Staubli VAL3: Robot_pippeting.dtx

aio aiAngleInclinarPipieta = {link=E954DA08-7D0C-47C0-8458-4D7DB0686071}
aio aiNumAmpolla = {link=F94C03B3-E86B-41EA-9D21-23C2AFB25672}
aio aiNumBanyera = {link=3DE16CC9-CC25-4818-8F3E-A7F806CB7947}
aio aiNumPipeta = {link=5259214B-6548-4F3D-A189-73563EE6598D}
aio aiNumPlacaDosi = {link=C4FBE503-E51F-4D58-BE10-749D221ACEB2}
aio aiProgramaPlc = {link=8E5652B8-E4D3-4267-ADD0-9C5A815DF2D8}
aio aiWordComPlc = {link=5C2A04D3-4005-4B43-8647-C0FC7B49D3AE}
aio aiXOffset = {link=95067B68-557B-4170-88AF-FC9CF5B8ED7A}
aio aiYOffset = {link=396181D2-5171-4A97-9799-32514BBB5F95}
aio aiZApro = {link=2D158B67-9924-4741-B554-50FB73F41045}
aio aiZOffset = {link=7513B562-B4FE-4098-AA1C-29A8706B731C}
aio aoForceJ1 = {link=9B11B2FE-99BA-4B55-9ED8-E4037A61E514}
aio aoForceJ2 = {link=DFC528C5-C573-4C02-A89E-35D8A1151078}
aio aoForceJ3 = {link=EC117CCB-E5D8-4A5C-AB6E-61FBA1760A17}
aio aoForceJ4 = {link=24340562-5DCA-47E3-A269-832024611405}
aio aoForceJ5 = {link=DB01A7CB-9BAD-4D46-B614-A585779504D9}
aio aoForceJ6 = {link=7A496CE7-D747-4637-B99A-202C76C7E7CC}
aio aoProgramaRobot = {link=5113B9A1-604C-4D8B-9163-7217CBF800C7}
aio aoStatusRobot = {link=F45B1EFD-4428-4D7D-8172-ECCCA511584C}
aio aoTascaAlarma = {link=53CEF201-0BB5-4BE1-8271-49FFF55CF52D}
aio aoWordComRobot = {link=6DF138BB-5CBA-4ACE-9C62-0AC3DF2353CB}
aio aoWorkingMode = {link=F7E03293-48A3-4B69-9598-2FE8DDFE0186}
aio aoXActual = {link=7FC267A8-BFA4-4039-BDA4-9FB4B4F71D48}
aio aoYActual = {link=E23CA4B2-A08C-4C00-8E97-94551E73BB09}
aio aoZActual = {link=78A73075-60CA-4FDB-AFF0-231125481CE1}
aio aoZonaHome = {link=F5709703-FBB2-4816-9A2C-2FC6F0D8F434}
bool bNewLog
bool bPrimerCicle
bool bTaskDone
dio diAlarmaPlc = {link=E7921EDF-610C-4E3F-84A7-2F1F4421B713}
dio diMarxaMaquina = {link=C1F67030-A9C1-420C-9B9B-1F49F7080557}
dio diSafetyRearme = {link=5367EF22-1F58-447B-AD12-D8B84F185C6B}
dio doAlarmaColisioRobot = {link=EA8AD671-7535-4BE0-BEBB-B9246DF094E3}
dio doAlarmaTascaRobot = {link=FCAEE04F-32B9-421A-B1DD-A8CEAA94D1C9}
dio doRobotEnMoviment = {link=B70DA9EE-8DF7-4C99-91DF-7149F2D942A3}
dio doRobotHome = {link=9957E281-FF01-4081-BA5E-7A249685580C}
dio doRobotPreparat = {link=19F8D819-A10B-480E-B6CD-15D2D35E2133}
dio doTaskDone = {link=0B0F13F6-DB8F-450C-AEE5-782BE1039C53}
frame fTaula = {fatherId=world[0]}
jointRx jHome = {j1=-3.455563, j2=6.0127238, j3=105.394535, j4=0.000031955, j5=68.591721, j6=-183.446968}
mdesc mAgafarPuntes = {accel=10, vel=10, decel=10, leave=0, reach=0}
mdesc mHome = {accel=25, vel=25, decel=25, leave=0, reach=0}
mdesc mLent = {accel=25, vel=25, decel=25, leave=10, reach=10}
mdesc mMig = {accel=50, vel=50, decel=50}
mdesc mNomSpeed
num nAngleInclinarPipeta
num nInerciaEina[3 3]
  [0,0] = 0.284
  [1,1] = 0.348
  [2,2] = 0.212
num nJointForce[6]
  [0] = 1.760942
  [1] = -21.676362
  [2] = -3.171848
  [3] = 1.641233
  [4] = -2.820579
  [5] = -0.389449
num nLog
num nPesEina = 15.8
num nSeqHome
num nWordComRobot = 6190
num nXOffset
num nYOffset
num nZApro = 50
num nZOffset
pointRx pAgafarPuntes1 = {x=287.432018, y=270.157151, z=-382.0291842, rx=179.996843, ry=-0.00380694, rz=0.700516, shoulder=lefty, elbow=epositive, wrist=wpositive, fatherId=fTaula[0]}
pointRx pAgafarPuntes8 = {x=285.860304, y=302.266054, z=-361.378441, rx=179.997149, ry=-0.00370527, rz=0.700442, shoulder=lefty, elbow=epositive, wrist=wpositive, fatherId=fTaula[0]}
pointRx pAmpolla[3]
  [0] = {x=493.522667, y=144.0778037, z=-386.621607, rx=179.997388, ry=-0.00407881, rz=0.700451, shoulder=lefty, elbow=epositive, wrist=wpositive, fatherId=fTaula[0]}
  [1] = {x=493.522667, y=144.0778037, z=-386.621607, rx=179.997388, ry=-0.00407881, rz=0.700451, shoulder=lefty, elbow=epositive, wrist=wpositive, fatherId=fTaula[0]}
  [2] = {x=546.605553, y=142.888702, z=-386.0523536, rx=179.997158, ry=-0.00493572, rz=0.700473, shoulder=lefty, elbow=epositive, wrist=wpositive, fatherId=fTaula[0]}
pointRx pBanyera[3]
  [0] = {x=336.466109, y=102.428458, z=-384.993166, rx=-0.00440943, ry=-179.995824, rz=-89.890495, shoulder=lefty, elbow=epositive, wrist=wpositive, fatherId=fTaula[0]}
  [1] = {x=336.466109, y=102.428458, z=-384.993166, rx=-0.00440943, ry=-179.995824, rz=-89.890495, shoulder=lefty, elbow=epositive, wrist=wpositive, fatherId=fTaula[0]}
  [2] = {x=336.466107, y=182.839383, z=-384.995018, rx=-0.003849, ry=-179.995539, rz=-89.890699, shoulder=lefty, elbow=epositive, wrist=wpositive, fatherId=fTaula[0]}
pointRx pDosi1[4]
  [0] = {x=305.52358, y=28.950334, z=-381.105899, rx=-0.00502749, ry=-179.983412, rz=-88.969574, shoulder=lefty, elbow=epositive, wrist=wpositive, fatherId=fTaula[0]}
  [1] = {x=305.523534, y=28.950368, z=-381.105899, rx=-0.00502365, ry=-179.983406, rz=-88.969579, shoulder=lefty, elbow=epositive, wrist=wpositive, fatherId=fTaula[0]}
  [2] = {x=306.96586, y=-130.963134, z=-381.122863, rx=-0.00532463, ry=-179.983113, rz=-88.9695, shoulder=lefty, elbow=epositive, wrist=wpositive, fatherId=fTaula[0]}
  [3] = {x=307.512874, y=-290.507285, z=-381.117547, rx=-0.00478912, ry=-179.98278, rz=-88.969551, shoulder=lefty, elbow=epositive, wrist=wpositive, fatherId=fTaula[0]}
pointRx pDosi8[4]
  [0] = {x=337.355483, y=31.174712, z=-385.0727918, rx=-0.0019009, ry=-179.993411, rz=-88.962152, shoulder=lefty, elbow=epositive, wrist=wpositive, fatherId=fTaula[0]}
  [1] = {x=337.355483, y=31.174712, z=-385.0727918, rx=-0.0019009, ry=-179.993411, rz=-88.962152, shoulder=lefty, elbow=epositive, wrist=wpositive, fatherId=fTaula[0]}
  [2] = {x=338.549957, y=-128.589669, z=-385.0544196, rx=0.000914256, ry=-179.993163, rz=-88.965193, shoulder=lefty, elbow=epositive, wrist=wpositive, fatherId=fTaula[0]}
  [3] = {x=339.326592, y=-288.609993, z=-385.0722156, rx=0.00206439, ry=-179.994818, rz=-88.964134, shoulder=lefty, elbow=epositive, wrist=wpositive, fatherId=fTaula[0]}
pointRx pHereHome = {x=172.623152, y=-333.816468, z=-286.331237, rx=0.00171927, ry=-179.997666, rz=-88.962057, shoulder=lefty, elbow=epositive, wrist=wpositive, fatherId=fTaula[0]}
pointRx pHome = {x=319.622111, y=0.736493, z=-179.743756, rx=180, shoulder=lefty, elbow=epositive, wrist=wpositive, fatherId=fTaula[0]}
pointRx pTirarPuntes = {x=172.623152, y=-333.816468, z=-336.331237, rx=0.00171927, ry=-179.997666, rz=-88.962057, shoulder=lefty, elbow=epositive, wrist=wpositive, fatherId=fTaula[0]}
string sLog[50]
  [1] = "1 - Inici: HOME"
  [2] = "17 - Fi: ANAR A APRO TIRAR PUNTES"
  [3] = "17 - Inici: ANAR A APRO TIRAR PUNTES"
  [4] = "18 - Fi: ANAR A TIRAR PUNTES"
  [5] = "18 - Inici: ANAR A TIRAR PUNTES"
  [6] = "17 - Fi: ANAR A APRO TIRAR PUNTES"
  [7] = "17 - Inici: ANAR A APRO TIRAR PUNTES"
  [8] = "20 - Fi: ANAR A APRO DOSI"
  [9] = "20 - Inici: ANAR A APRO DOSI"
  [10] = "22 - Fi: ANAR A POSICIONAT DOSI"
  [11] = "22 - Inici: ANAR A POSICIONAT DOSI"
  [12] = "21 - Fi: ANAR A DOSI"
  [13] = "21 - Inici: ANAR A DOSI"
  [14] = "20 - Fi: ANAR A APRO DOSI"
  [15] = "20 - Inici: ANAR A APRO DOSI"
  [16] = "20 - Fi: ANAR A APRO DOSI"
  [17] = "20 - Inici: ANAR A APRO DOSI"
  [18] = "22 - Fi: ANAR A POSICIONAT DOSI"
  [19] = "22 - Inici: ANAR A POSICIONAT DOSI"
  [20] = "21 - Fi: ANAR A DOSI"
  [21] = "21 - Inici: ANAR A DOSI"
  [22] = "20 - Fi: ANAR A APRO DOSI"
  [23] = "20 - Inici: ANAR A APRO DOSI"
  [24] = "20 - Fi: ANAR A APRO DOSI"
  [25] = "20 - Inici: ANAR A APRO DOSI"
  [26] = "21 - Fi: ANAR A DOSI"
  [27] = "21 - Inici: ANAR A DOSI"
  [28] = "20 - Fi: ANAR A APRO DOSI"
  [29] = "20 - Inici: ANAR A APRO DOSI"
  [30] = "15 - Fi: ANAR A APRO AGAFAR PUNTES"
  [31] = "15 - Inici: ANAR A APRO AGAFAR PUNTES"
  [32] = "16 - Fi: ANAR A AGAFAR PUNTES"
  [33] = "16 - Inici: ANAR A AGAFAR PUNTES"
  [34] = "15 - Fi: ANAR A APRO AGAFAR PUNTES"
  [35] = "15 - Inici: ANAR A APRO AGAFAR PUNTES"
  [36] = "17 - Fi: ANAR A APRO TIRAR PUNTES"
  [37] = "17 - Inici: ANAR A APRO TIRAR PUNTES"
  [38] = "18 - Fi: ANAR A TIRAR PUNTES"
  [39] = "18 - Inici: ANAR A TIRAR PUNTES"
  [40] = "17 - Fi: ANAR A APRO TIRAR PUNTES"
  [41] = "17 - Inici: ANAR A APRO TIRAR PUNTES"
  [42] = "20 - Fi: ANAR A APRO DOSI"
  [43] = "20 - Inici: ANAR A APRO DOSI"
  [44] = "22 - Fi: ANAR A POSICIONAT DOSI"
  [45] = "22 - Inici: ANAR A POSICIONAT DOSI"
  [46] = "21 - Fi: ANAR A DOSI"
  [47] = "21 - Inici: ANAR A DOSI"
  [48] = "20 - Fi: ANAR A APRO DOSI"
  [49] = "20 - Inici: ANAR A APRO DOSI"
string sNewLog = "1 - Fi: HOME"
tool tToolActiva = {z=285, fatherId=flange[0]}
tool tToolPipeta1 = {z=300, fatherId=flange[0]}
tool tToolPipeta8 = {z=285, fatherId=flange[0]}
trsf trEina = {x=94.8, y=-0.4, z=220.5}
